Fanuc KAREL source: kt00573.KL

-- PROVISIONAL review KL for V1013-1; original PC SHA256 e396e45302b17937652401cee1ce982f2cbfbd569fa35166107c885ea25c33ed
-- Incomplete behavior may be omitted. Consult companion uncertainty JSON. Do not deploy.
PROGRAM KT00573
%NOLOCKGROUP
VAR
  R1 : REAL
-- UNRESOLVED_DECL V2 type=000013
-- UNRESOLVED_DECL OUT type=000013
BEGIN
  -- UNRESOLVED_PC offsets 5-16; opcodes 2E,23
  -- UNRESOLVED_PC offsets 21-36; opcodes 2E,22,32,35
  -- UNRESOLVED_PC offsets 41-63; opcodes 21,49,8C,4A
  -- UNRESOLVED_PC offsets 68-72; opcodes 7F
END KT00573
